PROGRAM PRG_FB_AnalogOutput_Test
VAR
	bFirsCycle		: BOOL := TRUE;		(* First cycle flag *)
	rValue			: REAL;				(* Scaled value that is send to channel *)
	
	rValueMin 		: REAL := 0.0;		(*  *)
	rValueMax		: REAL := 10.0;		(*  *)
	rChannelMin		: REAL := 0.0;		(*  *)
	rChannelMax		: REAL := 32767.0;	(*  *)
	
	fbAnalogOutput	: FB_AnalogOutput;	(* Analog input object *)
END_VAR

(* Set properties *)
IF bFirsCycle THEN
	bFirsCycle := FALSE;
	fbAnalogOutput.MR_FirstCycle( 	sName 			:= 'My test analog output',
									rValueScaledMin := rValueMin,
									rValueScaledMax := rValueMax,
									rChannelMin 	:= rChannelMin,
									rChannelMax		:= rChannelMax);
END_IF

(* Cyclic properties update *)
fbAnalogOutput.ChannelMin	:= rChannelMin;
fbAnalogOutput.ChannelMax 	:= rChannelMax;
fbAnalogOutput.ValueMin 	:= rValueMin;
fbAnalogOutput.ValueMax 	:= rValueMax;

(* Send value to channel *)
fbAnalogOutput.Value 		:= rValue;
fbAnalogOutput();

END_PROGRAM

(* stored: Version 1.1.0.1, ProductVersion 3.1.4024.9
   POU PRG_FB_AnalogOutput_Test: Id {4a2c79c5-ff77-4eb8-8ed2-f0a08b6d6ada}, SpecialFunc None *)
